// Mitsubishi GX Works2 project: PLC 특수기능 (SET, RST)   PLC: Q03UDV

PROGRAM MAIN
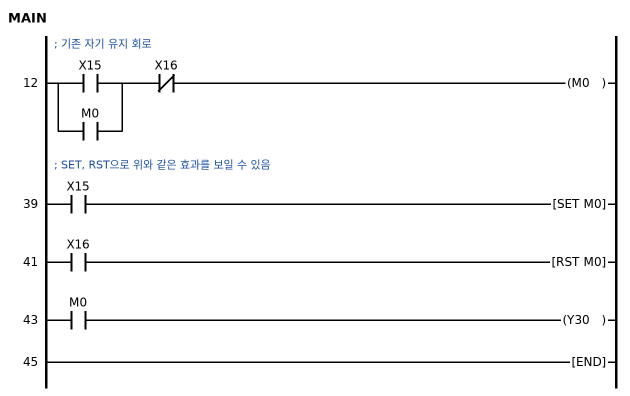
; 기존 자기 유지 회로
12    LD      X15
      OR      M0
      ANI     X16
      OUT     M0
; SET, RST으로 위와 같은 효과를 보일 수 있음
39    LD      X15
      SET     M0
41    LD      X16
      RST     M0
43    LD      M0
      OUT     Y30
45    END
END_PROGRAM
